FUNCTION_BLOCK XtsEnableSequence EXTENDS TaskBase
VAR_INPUT
END_VAR
VAR_OUTPUT
END_VAR
VAR
	_collisionGroup : ICollisionGroup;
	addMover : AddMoverToGroupTask(_collisionGroup);
	moverNumbers : UINT;
	AllMoversEnabled: BOOL;
	EnableTrigger : BOOL;	
	Logger : TcMessage_Ext;
	arrMovers : ARRAY[1..SystemParameters.NumberOfMovers] OF IMover;
END_VAR

{analysis -2}

METHOD Abort : BOOL
EnableTrigger := FALSE;
State := 0;
addMover.Abort();
END_METHOD

METHOD Cycle : HRESULT
VAR_INPUT
END_VAR
Cycle := S_OK;
CASE State OF
	0:
		IF EnableTrigger THEN
			Cycle := S_PENDING;
			State := 10;
			EnableTrigger := FALSE;
			moverNumbers := 1;
			_Busy := TRUE;
			_Done := FALSE;
			_Error := FALSE;
		END_IF
		
	10:
		FOR moverNumbers := 1 TO SystemParameters.NumberOfMovers DO
			arrMovers[moverNumbers].ResetAxis();
		END_FOR
		moverNumbers := 1;
		State := 20;
		
	20:
		IF _collisionGroup.GroupState = CAGroupStatus.mcGroupStateErrorStop THEN
			_collisionGroup.Reset();
			Logger.Send(TC_EVENTS.XtsCaGroupEvents.CAGroupReset,'');
		END_IF
		State := 30;
		
	30:
		arrMovers[moverNumbers].IdentInGroup := UINT_TO_INT( moverNumbers);
		addMover.AddMover(MoverToAdd := arrMovers[moverNumbers]);
		Logger.Send(TC_EVENTS.XtsCaGroupEvents.AddingMoverToGroup,UINT_TO_STRING(moverNumbers));
		State := 40;
		
	40:
		IF addMover.Done THEN
			IF moverNumbers <> SystemParameters.NumberOfMovers THEN
				moverNumbers := moverNumbers + 1;
				State := 30;
			ELSE
				Logger.Send(TC_EVENTS.XtsCaGroupEvents.AllMoversAdded,'');
				FOR moverNumbers := 1 TO SystemParameters.NumberOfMovers DO
					arrMovers[moverNumbers].EnableAxis();
				END_FOR
				State := 50;
			END_IF
		END_IF
		
	50:
		AllMoversEnabled := TRUE;
		FOR moverNumbers := 1 TO SystemParameters.NumberOfMovers DO
			AllMoversEnabled := TRUE AND arrMovers[moverNumbers].isEnabled();
		END_FOR
		IF AllMoversEnabled THEN
			Logger.Send(TC_EVENTS.XtsCaGroupEvents.AllMoversEnabled,'');
			_collisionGroup.Enable();
			Logger.Send(TC_EVENTS.XtsCaGroupEvents.CAGroupEnable,'');
			State := 60;
		END_IF
		
	60:
		IF _collisionGroup.GroupState = 2 THEN
			State := 0;
			_Busy := FALSE;
			_Done := TRUE;
			Cycle := S_PENDING;
		END_IF
	ELSE
		Cycle := E_FAIL;
END_CASE

addMover.Cycle();
END_METHOD

METHOD Enable : BOOL
VAR_INPUT
END_VAR
IF NOT _Busy THEN
	EnableTrigger := Enable := true;
END_IF
END_METHOD

METHOD FB_init : BOOL
VAR_INPUT
	bInitRetains : BOOL; // if TRUE, the retain variables are initialized (warm start / cold start)
	bInCopyCode : BOOL;  // if TRUE, the instance afterwards gets moved into the copy code (online change)
	MyCaGroup : ICollisionGroup;
END_VAR
_collisionGroup := MyCaGroup;
addMover.FB_init(FALSE, FALSE, myCaGroup);
END_METHOD

PROPERTY MoverArray : array[1..SystemParameters.NumberOfMovers] of IMover
GET
MoverArray := arrMovers;
END_GET
SET
arrMovers := MoverArray;
END_SET
END_PROPERTY

END_FUNCTION_BLOCK

(* stored: Version 1.1.0.1, ProductVersion 3.1.4024.12
   POU XtsEnableSequence: Id {b7e7ab09-3a30-4ddb-a242-e0b5aa00cbc9}, SpecialFunc None
   Method Abort: Id {9cec9788-9ce4-4a9f-821c-172bdb3141aa}
   Method Cycle: Id {2913b891-dfae-43d9-b9d3-4a1a1101f452}
   Method Enable: Id {1c2a3468-bb52-4165-8d13-732b960a1dd0}
   Method FB_init: Id {a4125f89-7eca-48c2-8cb0-d4574c798d78}
   Property MoverArray: Id {2acddb92-7228-4ce1-abf4-c52047e8db87}
   Get Get: Id {45d4b80a-6470-4599-bc0b-107c251d2b9f}
   Set Set: Id {2f5a4b68-8d6e-4eaa-8b71-147268b7ef4e} *)
